Staubli VAL3: ActionItem.pjx

--- ActionItem.pjx ---
Parameters version=s7.2.1 stackSize=5000 millimeterUnit=true
Data file=ActionItem.dtx
Type name=InstrItem path=Disk://kernel/template/InstrItem/InstrItem.pjx
Type name=Trajectory path=Disk://kernel/template/Trajectory/Trajectory.pjx

--- ActionItem.dtx ---
public num nDistance
public num nMoveId
public num nTimeId
public num nPointId
public InstrItem iInstr[3]
  [0]
    string sType
    string sData
  [1]
    string sType
    string sData
  [2]
    string sType
    string sData
public string sIdTraj
